INTERFACE I_LensSetCompounder EXTENDS I_Fallible


METHOD Compound : LREAL
VAR_INPUT
    fFocalLength : LREAL;
    fSourceDistance : LREAL;
END_VAR
END_METHOD


PROPERTY FocalLengthCompounded : LREAL
GET
END_GET
END_PROPERTY


METHOD Reset
END_METHOD

END_INTERFACE

(* stored: Version 1.1.0.1
   Itf I_LensSetCompounder: Id {3bb8a747-47ad-48be-9f6b-bd8d2a64ee36}
   Method Compound: Id {10181a56-66cb-4ee4-86a4-1ee71e6ce912}
   Property FocalLengthCompounded: Id {a699a99b-cdeb-4edc-9aba-ff0abe45dff8}
   Get Get: Id {1bff1399-2255-4356-8b0e-46b81527c1de}
   Method Reset: Id {b8f90921-d231-4706-a1d2-5c3ccbdb351f} *)
